TYPE OP130_Recipe :
STRUCT


END_STRUCT
END_TYPE

(* stored: Version 1.1.0.1, ProductVersion 3.1.4024.11
   DUT OP130_Recipe: Id {755cc43e-248b-436a-b935-19d241abc29e} *)
